Staubli VAL3: remote_isHome.pgx

program remote_isHome()
  local joint l_jHere
  local num l_nResult
  local num l_nSize
  local string l_sItem
begin
  // look if home was loaded
  if (!cycleStatus:bHomeLoaded or jHome:libPath()=="" or find(jHome:libPath(),"template")!=-1) and saveData:bToReload==false
    call remote_loadHome(l_nResult)
  endIf
  // ok home is in the ram
  l_sItem="home"
  l_nSize=size(jHome:tTraj[l_sItem].tData)-1
  if l_nResult==0 and jHome:tTraj[l_sItem].tData[l_nSize].jJoint!={0,0,0,0,0,0}
    // check if the the robot is nearby
    if abs(herej()-jHome:tTraj[l_sItem].tData[l_nSize].jJoint)<{1,1,1,2,2,2}
      // the robot is at home
      cycleStatus:bIsHome=true
    else
      cycleStatus:bIsHome=false
    endIf
  else
    cycleStatus:bIsHome=false
  endIf
  //
end
